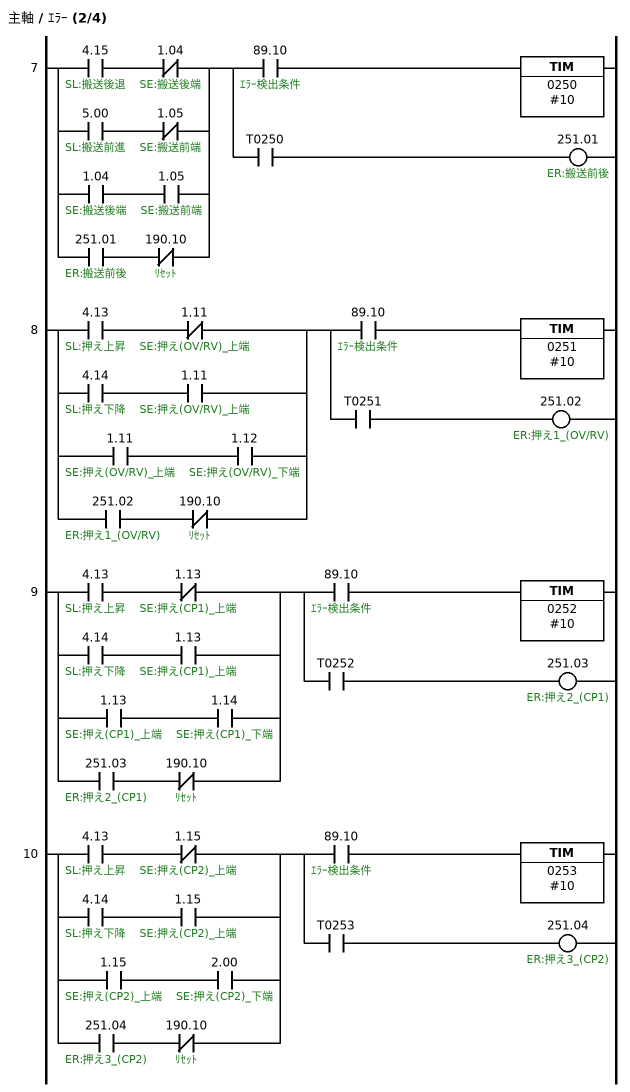
; rung 7
LD 4.15  ; SL:搬送後退
ANDNOT 1.04  ; SE:搬送後端
LD 5.00  ; SL:搬送前進
ANDNOT 1.05  ; SE:搬送前端
ORLD
LD 1.04  ; SE:搬送後端
AND 1.05  ; SE:搬送前端
ORLD
LD 251.01  ; ER:搬送前後
ANDNOT 190.10  ; ﾘｾｯﾄ
ORLD
OUT TR0
AND 89.10  ; ｴﾗｰ検出条件
TIM 0250 #10
LD TR0
AND T0250
OUT 251.01  ; ER:搬送前後
; rung 8
LD 4.13  ; SL:押え上昇
ANDNOT 1.11  ; SE:押え(OV/RV)_上端
LD 4.14  ; SL:押え下降
AND 1.11  ; SE:押え(OV/RV)_上端
ORLD
LD 1.11  ; SE:押え(OV/RV)_上端
AND 1.12  ; SE:押え(OV/RV)_下端
ORLD
LD 251.02  ; ER:押え1_(OV/RV)
ANDNOT 190.10  ; ﾘｾｯﾄ
ORLD
OUT TR0
AND 89.10  ; ｴﾗｰ検出条件
TIM 0251 #10
LD TR0
AND T0251
OUT 251.02  ; ER:押え1_(OV/RV)
; rung 9
LD 4.13  ; SL:押え上昇
ANDNOT 1.13  ; SE:押え(CP1)_上端
LD 4.14  ; SL:押え下降
AND 1.13  ; SE:押え(CP1)_上端
ORLD
LD 1.13  ; SE:押え(CP1)_上端
AND 1.14  ; SE:押え(CP1)_下端
ORLD
LD 251.03  ; ER:押え2_(CP1)
ANDNOT 190.10  ; ﾘｾｯﾄ
ORLD
OUT TR0
AND 89.10  ; ｴﾗｰ検出条件
TIM 0252 #10
LD TR0
AND T0252
OUT 251.03  ; ER:押え2_(CP1)
; rung 10
LD 4.13  ; SL:押え上昇
ANDNOT 1.15  ; SE:押え(CP2)_上端
LD 4.14  ; SL:押え下降
AND 1.15  ; SE:押え(CP2)_上端
ORLD
LD 1.15  ; SE:押え(CP2)_上端
AND 2.00  ; SE:押え(CP2)_下端
ORLD
LD 251.04  ; ER:押え3_(CP2)
ANDNOT 190.10  ; ﾘｾｯﾄ
ORLD
OUT TR0
AND 89.10  ; ｴﾗｰ検出条件
TIM 0253 #10
LD TR0
AND T0253
OUT 251.04  ; ER:押え3_(CP2)

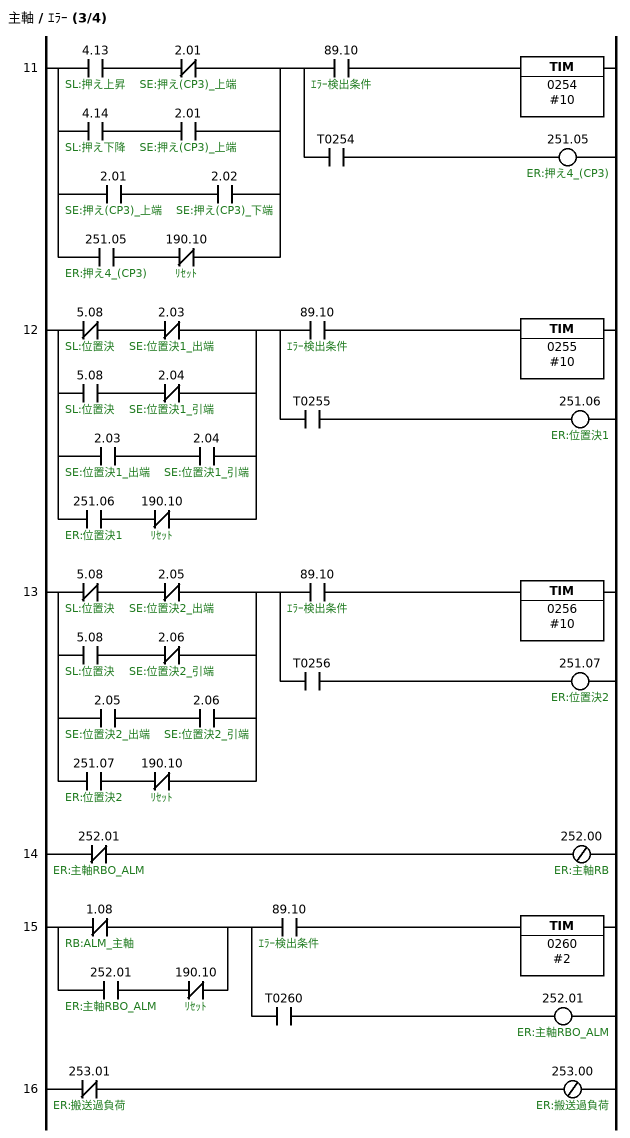
; rung 11
LD 4.13  ; SL:押え上昇
ANDNOT 2.01  ; SE:押え(CP3)_上端
LD 4.14  ; SL:押え下降
AND 2.01  ; SE:押え(CP3)_上端
ORLD
LD 2.01  ; SE:押え(CP3)_上端
AND 2.02  ; SE:押え(CP3)_下端
ORLD
LD 251.05  ; ER:押え4_(CP3)
ANDNOT 190.10  ; ﾘｾｯﾄ
ORLD
OUT TR0
AND 89.10  ; ｴﾗｰ検出条件
TIM 0254 #10
LD TR0
AND T0254
OUT 251.05  ; ER:押え4_(CP3)
; rung 12
LDNOT 5.08  ; SL:位置決
ANDNOT 2.03  ; SE:位置決1_出端
LD 5.08  ; SL:位置決
ANDNOT 2.04  ; SE:位置決1_引端
ORLD
LD 2.03  ; SE:位置決1_出端
AND 2.04  ; SE:位置決1_引端
ORLD
LD 251.06  ; ER:位置決1
ANDNOT 190.10  ; ﾘｾｯﾄ
ORLD
OUT TR0
AND 89.10  ; ｴﾗｰ検出条件
TIM 0255 #10
LD TR0
AND T0255
OUT 251.06  ; ER:位置決1
; rung 13
LDNOT 5.08  ; SL:位置決
ANDNOT 2.05  ; SE:位置決2_出端
LD 5.08  ; SL:位置決
ANDNOT 2.06  ; SE:位置決2_引端
ORLD
LD 2.05  ; SE:位置決2_出端
AND 2.06  ; SE:位置決2_引端
ORLD
LD 251.07  ; ER:位置決2
ANDNOT 190.10  ; ﾘｾｯﾄ
ORLD
OUT TR0
AND 89.10  ; ｴﾗｰ検出条件
TIM 0256 #10
LD TR0
AND T0256
OUT 251.07  ; ER:位置決2
; rung 14
LDNOT 252.01  ; ER:主軸RBO_ALM
OUTNOT 252.00  ; ER:主軸RB
; rung 15
LDNOT 1.08  ; RB:ALM_主軸
LD 252.01  ; ER:主軸RBO_ALM
ANDNOT 190.10  ; ﾘｾｯﾄ
ORLD
OUT TR0
AND 89.10  ; ｴﾗｰ検出条件
TIM 0260 #2
LD TR0
AND T0260
OUT 252.01  ; ER:主軸RBO_ALM
; rung 16
LDNOT 253.01  ; ER:搬送過負荷
OUTNOT 253.00  ; ER:搬送過負荷

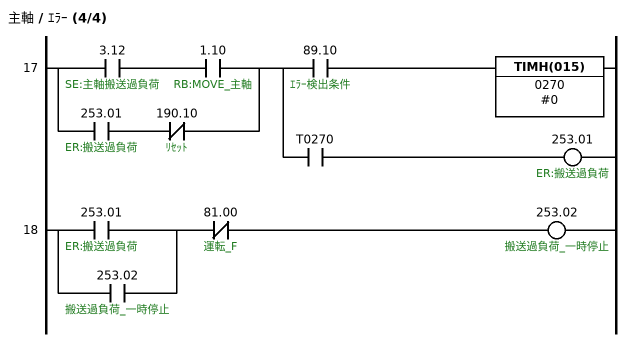
; rung 17
LD 3.12  ; SE:主軸搬送過負荷
AND 1.10  ; RB:MOVE_主軸
LD 253.01  ; ER:搬送過負荷
ANDNOT 190.10  ; ﾘｾｯﾄ
ORLD
OUT TR0
AND 89.10  ; ｴﾗｰ検出条件
TIMH(015) 0270 #0
LD TR0
AND T0270
OUT 253.01  ; ER:搬送過負荷
; rung 18
LD 253.01  ; ER:搬送過負荷
OR 253.02  ; 搬送過負荷_一時停止
ANDNOT 81.00  ; 運転_F
OUT 253.02  ; 搬送過負荷_一時停止

### Section END
; rung 0
END(001)

## Program 供給 (cyclic task 3)

### Section 制御

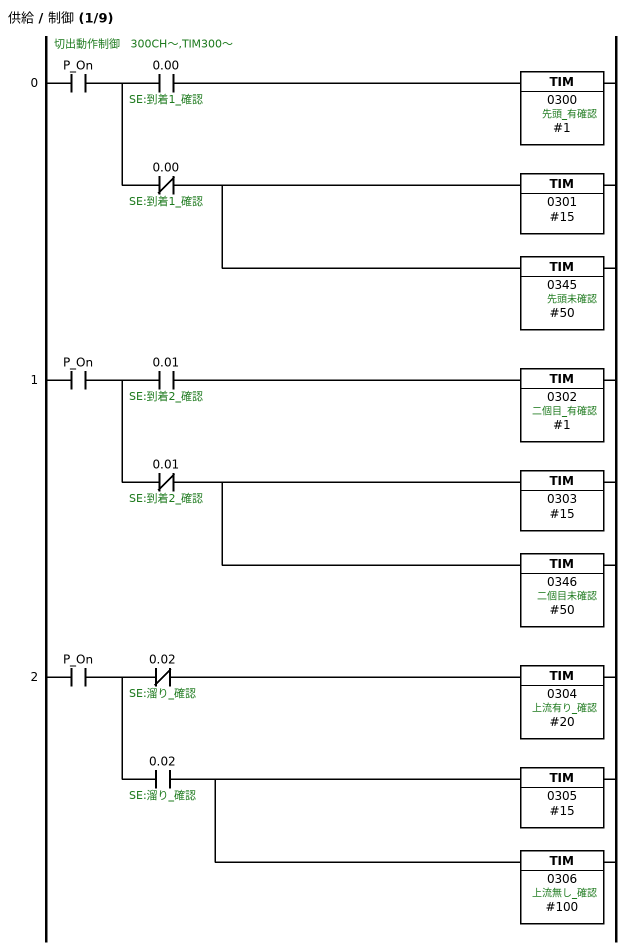
; rung 0: 切出動作制御   300CH～,TIM300～
LD P_On
OUT TR0
AND 0.00  ; SE:到着1_確認
TIM 0300 #1  ; 先頭_有確認
LD TR0
ANDNOT 0.00  ; SE:到着1_確認
TIM 0301 #15
TIM 0345 #50  ; 先頭未確認
; rung 1
LD P_On
OUT TR0
AND 0.01  ; SE:到着2_確認
TIM 0302 #1  ; 二個目_有確認
LD TR0
ANDNOT 0.01  ; SE:到着2_確認
TIM 0303 #15
TIM 0346 #50  ; 二個目未確認
; rung 2
LD P_On
OUT TR0
ANDNOT 0.02  ; SE:溜り_確認
TIM 0304 #20  ; 上流有り_確認
LD TR0
AND 0.02  ; SE:溜り_確認
TIM 0305 #15
TIM 0306 #100  ; 上流無し_確認

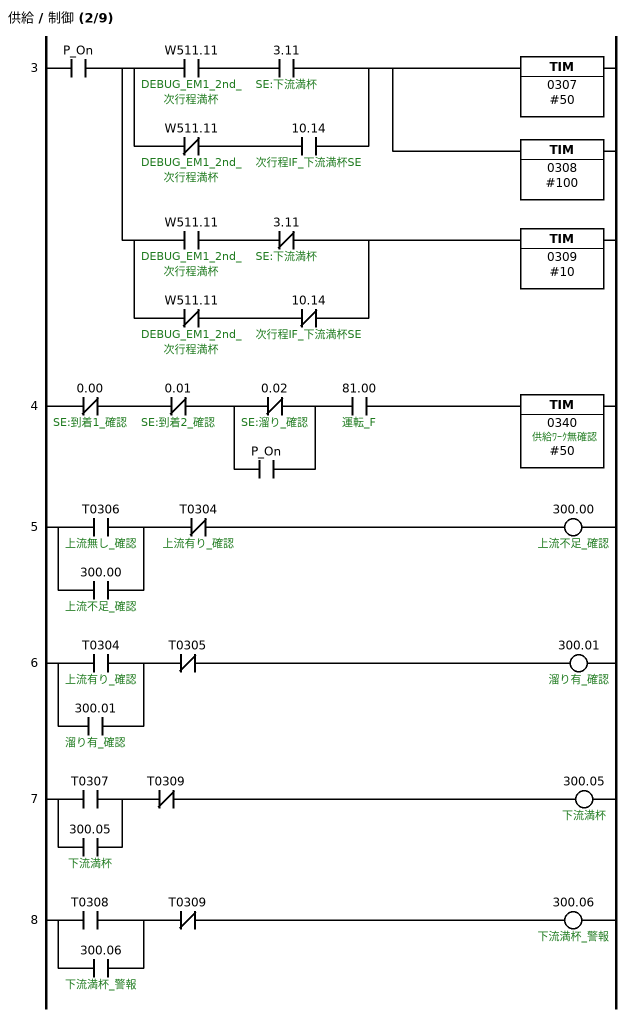
; rung 3
LD P_On
OUT TR0
LD W511.11  ; DEBUG_EM1_2nd_次行程満杯
AND 3.11  ; SE:下流満杯
LDNOT W511.11  ; DEBUG_EM1_2nd_次行程満杯
AND 10.14  ; 次行程IF_下流満杯SE
ORLD
ANDLD
TIM 0307 #50
TIM 0308 #100
LD TR0
LD W511.11  ; DEBUG_EM1_2nd_次行程満杯
ANDNOT 3.11  ; SE:下流満杯
LDNOT W511.11  ; DEBUG_EM1_2nd_次行程満杯
ANDNOT 10.14  ; 次行程IF_下流満杯SE
ORLD
ANDLD
TIM 0309 #10
; rung 4
LDNOT 0.00  ; SE:到着1_確認
ANDNOT 0.01  ; SE:到着2_確認
LDNOT 0.02  ; SE:溜り_確認
OR P_On
ANDLD
AND 81.00  ; 運転_F
TIM 0340 #50  ; 供給ﾜｰｸ無確認
; rung 5
LD T0306  ; 上流無し_確認
OR 300.00  ; 上流不足_確認
ANDNOT T0304  ; 上流有り_確認
OUT 300.00  ; 上流不足_確認
; rung 6
LD T0304  ; 上流有り_確認
OR 300.01  ; 溜り有_確認
ANDNOT T0305
OUT 300.01  ; 溜り有_確認
; rung 7
LD T0307
OR 300.05  ; 下流満杯
ANDNOT T0309
OUT 300.05  ; 下流満杯
; rung 8
LD T0308
OR 300.06  ; 下流満杯_警報
ANDNOT T0309
OUT 300.06  ; 下流満杯_警報

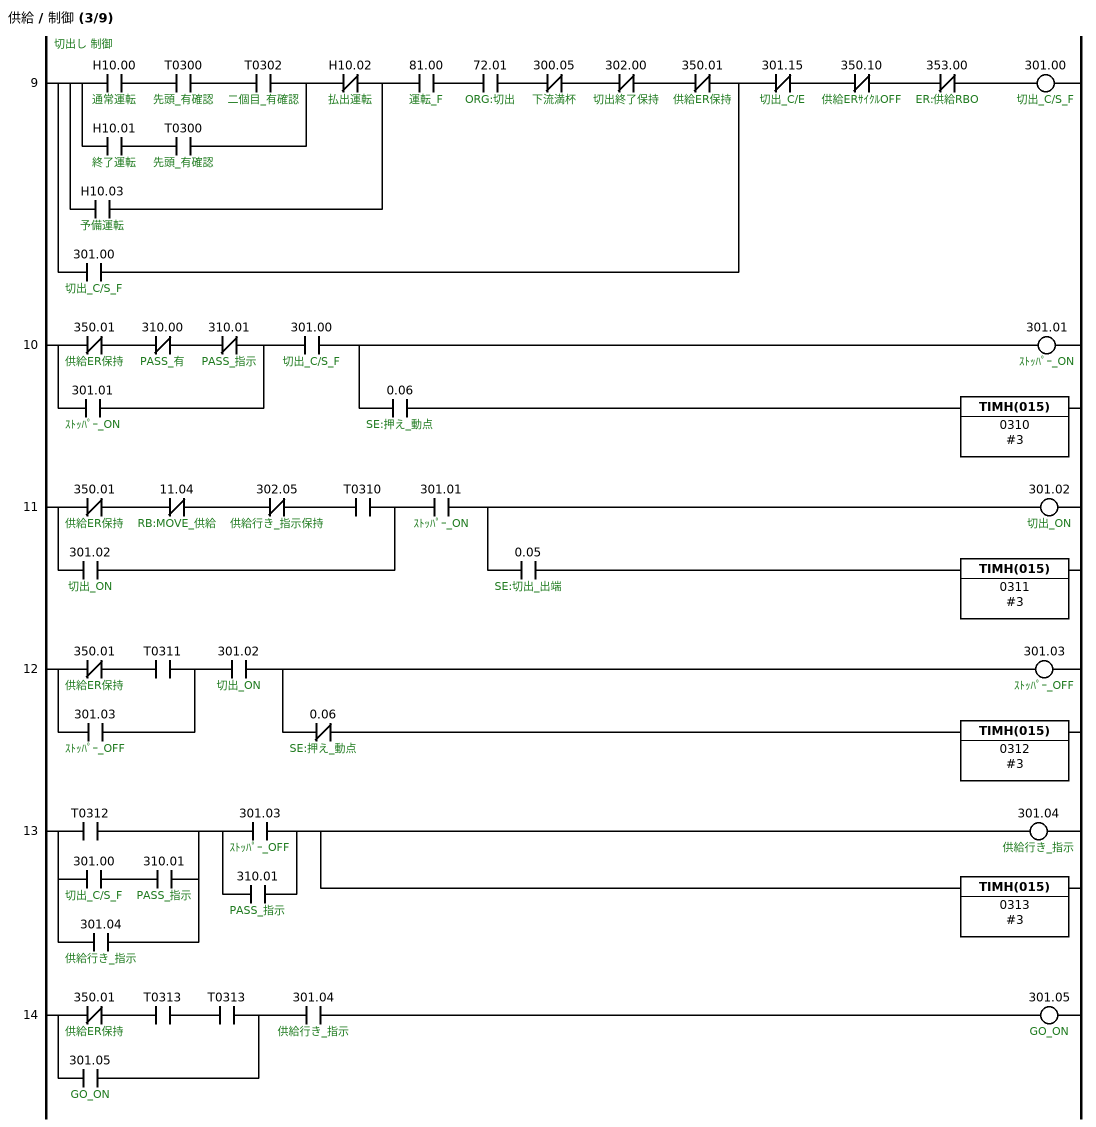
; rung 9: 切出し 制御
LD H10.00  ; 通常運転
AND T0300  ; 先頭_有確認
AND T0302  ; 二個目_有確認
LD H10.01  ; 終了運転
AND T0300  ; 先頭_有確認
ORLD
ANDNOT H10.02  ; 払出運転
OR H10.03  ; 予備運転
AND 81.00  ; 運転_F
AND 72.01  ; ORG:切出
ANDNOT 300.05  ; 下流満杯
ANDNOT 302.00  ; 切出終了保持
ANDNOT 350.01  ; 供給ER保持
OR 301.00  ; 切出_C/S_F
ANDNOT 301.15  ; 切出_C/E
ANDNOT 350.10  ; 供給ERｻｲｸﾙOFF
ANDNOT 353.00  ; ER:供給RBO
OUT 301.00  ; 切出_C/S_F
; rung 10
LDNOT 350.01  ; 供給ER保持
ANDNOT 310.00  ; PASS_有
ANDNOT 310.01  ; PASS_指示
OR 301.01  ; ｽﾄｯﾊﾟｰ_ON
AND 301.00  ; 切出_C/S_F
OUT 301.01  ; ｽﾄｯﾊﾟｰ_ON
AND 0.06  ; SE:押え_動点
TIMH(015) 0310 #3
; rung 11
LDNOT 350.01  ; 供給ER保持
ANDNOT 11.04  ; RB:MOVE_供給
ANDNOT 302.05  ; 供給行き_指示保持
AND T0310
OR 301.02  ; 切出_ON
AND 301.01  ; ｽﾄｯﾊﾟｰ_ON
OUT 301.02  ; 切出_ON
AND 0.05  ; SE:切出_出端
TIMH(015) 0311 #3
; rung 12
LDNOT 350.01  ; 供給ER保持
AND T0311
OR 301.03  ; ｽﾄｯﾊﾟｰ_OFF
AND 301.02  ; 切出_ON
OUT 301.03  ; ｽﾄｯﾊﾟｰ_OFF
ANDNOT 0.06  ; SE:押え_動点
TIMH(015) 0312 #3
; rung 13
LD T0312
LD 301.00  ; 切出_C/S_F
AND 310.01  ; PASS_指示
ORLD
OR 301.04  ; 供給行き_指示
LD 301.03  ; ｽﾄｯﾊﾟｰ_OFF
OR 310.01  ; PASS_指示
ANDLD
OUT 301.04  ; 供給行き_指示
TIMH(015) 0313 #3
; rung 14
LDNOT 350.01  ; 供給ER保持
AND T0313
AND T0313
OR 301.05  ; GO_ON
AND 301.04  ; 供給行き_指示
OUT 301.05  ; GO_ON

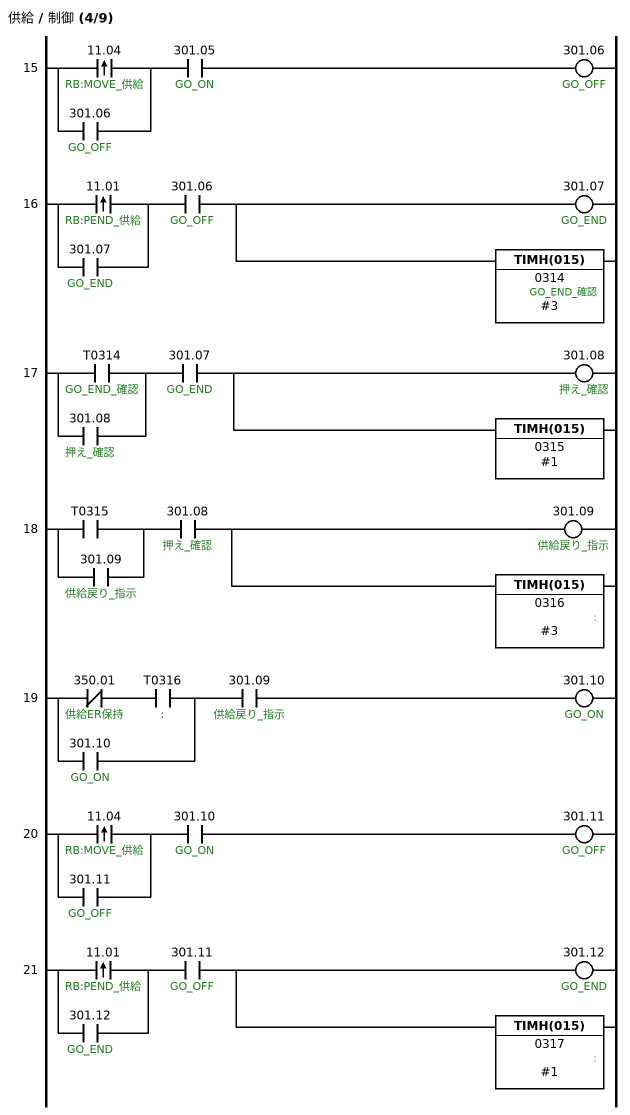
; rung 15
@LD 11.04  ; RB:MOVE_供給
OR 301.06  ; GO_OFF
AND 301.05  ; GO_ON
OUT 301.06  ; GO_OFF
; rung 16
@LD 11.01  ; RB:PEND_供給
OR 301.07  ; GO_END
AND 301.06  ; GO_OFF
OUT 301.07  ; GO_END
TIMH(015) 0314 #3  ; GO_END_確認
; rung 17
LD T0314  ; GO_END_確認
OR 301.08  ; 押え_確認
AND 301.07  ; GO_END
OUT 301.08  ; 押え_確認
TIMH(015) 0315 #1
; rung 18
LD T0315
OR 301.09  ; 供給戻り_指示
AND 301.08  ; 押え_確認
OUT 301.09  ; 供給戻り_指示
TIMH(015) 0316 #3  ; :
; rung 19
LDNOT 350.01  ; 供給ER保持
AND T0316  ; :
OR 301.10  ; GO_ON
AND 301.09  ; 供給戻り_指示
OUT 301.10  ; GO_ON
; rung 20
@LD 11.04  ; RB:MOVE_供給
OR 301.11  ; GO_OFF
AND 301.10  ; GO_ON
OUT 301.11  ; GO_OFF
; rung 21
@LD 11.01  ; RB:PEND_供給
OR 301.12  ; GO_END
AND 301.11  ; GO_OFF
OUT 301.12  ; GO_END
TIMH(015) 0317 #1  ; :

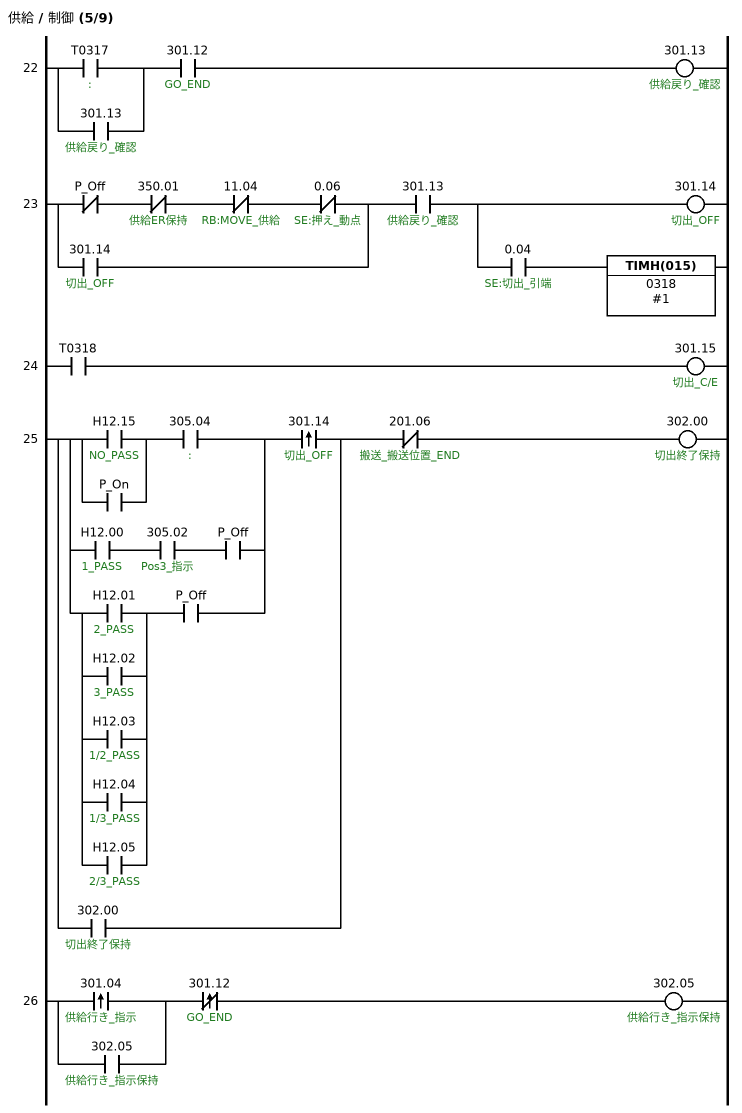
; rung 22
LD T0317  ; :
OR 301.13  ; 供給戻り_確認
AND 301.12  ; GO_END
OUT 301.13  ; 供給戻り_確認
; rung 23
LDNOT P_Off
ANDNOT 350.01  ; 供給ER保持
ANDNOT 11.04  ; RB:MOVE_供給
ANDNOT 0.06  ; SE:押え_動点
OR 301.14  ; 切出_OFF
AND 301.13  ; 供給戻り_確認
OUT 301.14  ; 切出_OFF
AND 0.04  ; SE:切出_引端
TIMH(015) 0318 #1
; rung 24
LD T0318
OUT 301.15  ; 切出_C/E
; rung 25
LD H12.15  ; NO_PASS
OR P_On
AND 305.04  ; :
LD H12.00  ; 1_PASS
AND 305.02  ; Pos3_指示
AND P_Off
ORLD
LD H12.01  ; 2_PASS
OR H12.02  ; 3_PASS
OR H12.03  ; 1/2_PASS
OR H12.04  ; 1/3_PASS
OR H12.05  ; 2/3_PASS
AND P_Off
ORLD
@AND 301.14  ; 切出_OFF
OR 302.00  ; 切出終了保持
ANDNOT 201.06  ; 搬送_搬送位置_END
OUT 302.00  ; 切出終了保持
; rung 26
@LD 301.04  ; 供給行き_指示
OR 302.05  ; 供給行き_指示保持
@ANDNOT 301.12  ; GO_END
OUT 302.05  ; 供給行き_指示保持

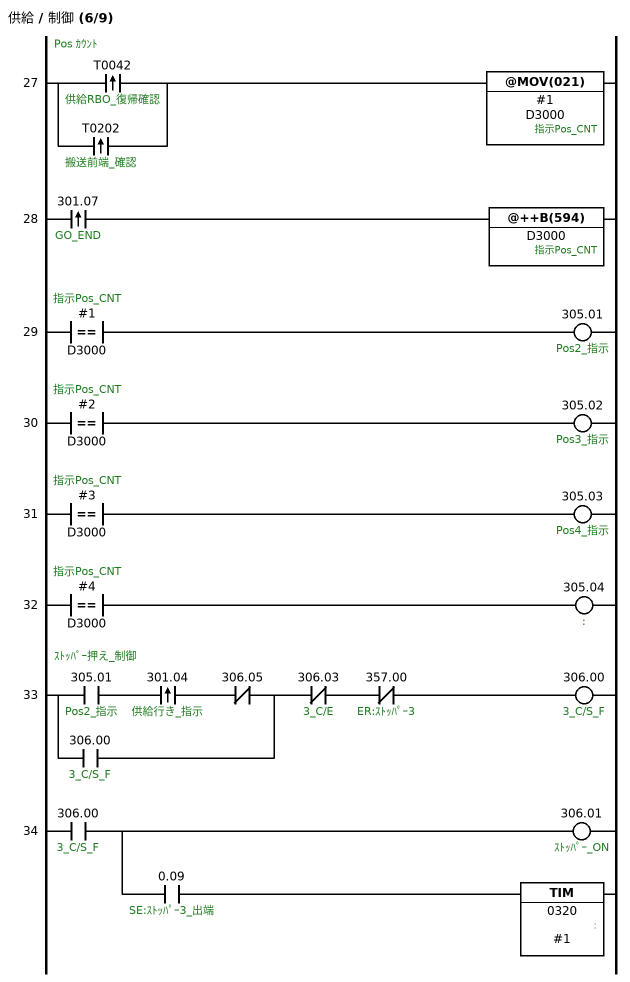
; rung 27: Pos ｶｳﾝﾄ
@LD T0042  ; 供給RBO_復帰確認
@OR T0202  ; 搬送前端_確認
@MOV(021) #1 D3000  ; 指示Pos_CNT
; rung 28
@LD 301.07  ; GO_END
@++B(594) D3000  ; 指示Pos_CNT
; rung 29
LD=(300) #1 D3000  ; 指示Pos_CNT
OUT 305.01  ; Pos2_指示
; rung 30
LD=(300) #2 D3000  ; 指示Pos_CNT
OUT 305.02  ; Pos3_指示
; rung 31
LD=(300) #3 D3000  ; 指示Pos_CNT
OUT 305.03  ; Pos4_指示
; rung 32
LD=(300) #4 D3000  ; 指示Pos_CNT
OUT 305.04  ; :
; rung 33: ｽﾄｯﾊﾟｰ押え_制御
LD 305.01  ; Pos2_指示
@AND 301.04  ; 供給行き_指示
ANDNOT 306.05
OR 306.00  ; 3_C/S_F
ANDNOT 306.03  ; 3_C/E
ANDNOT 357.00  ; ER:ｽﾄｯﾊﾟｰ3
OUT 306.00  ; 3_C/S_F
; rung 34
LD 306.00  ; 3_C/S_F
OUT 306.01  ; ｽﾄｯﾊﾟｰ_ON
AND 0.09  ; SE:ｽﾄｯﾊﾟｰ3_出端
TIM 0320 #1  ; :

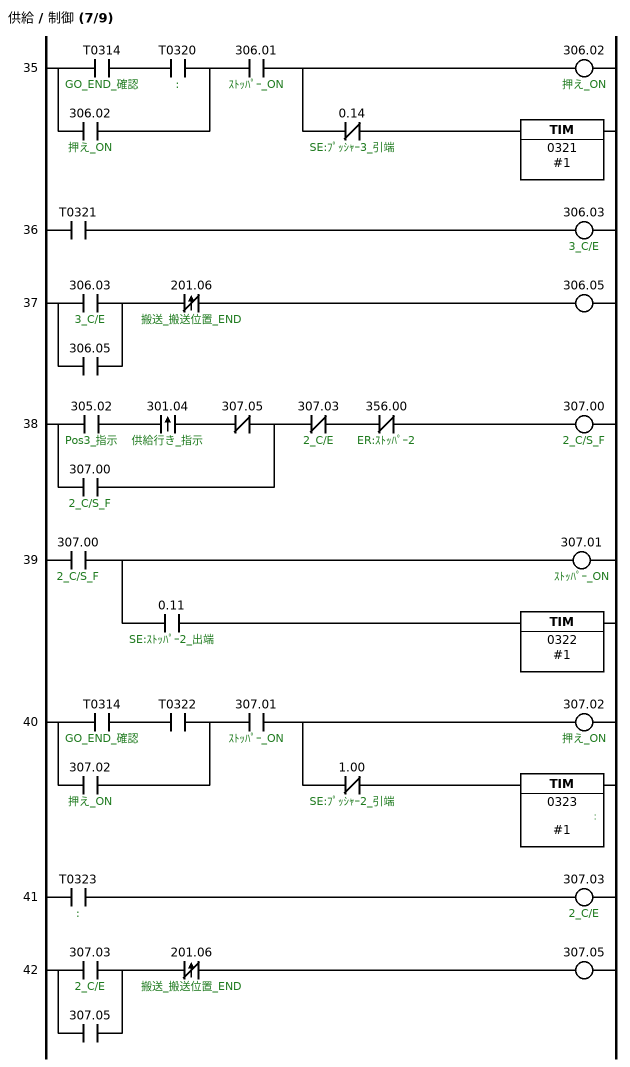
; rung 35
LD T0314  ; GO_END_確認
AND T0320  ; :
OR 306.02  ; 押え_ON
AND 306.01  ; ｽﾄｯﾊﾟｰ_ON
OUT 306.02  ; 押え_ON
ANDNOT 0.14  ; SE:ﾌﾟｯｼｬｰ3_引端
TIM 0321 #1
; rung 36
LD T0321
OUT 306.03  ; 3_C/E
; rung 37
LD 306.03  ; 3_C/E
OR 306.05
@ANDNOT 201.06  ; 搬送_搬送位置_END
OUT 306.05
; rung 38
LD 305.02  ; Pos3_指示
@AND 301.04  ; 供給行き_指示
ANDNOT 307.05
OR 307.00  ; 2_C/S_F
ANDNOT 307.03  ; 2_C/E
ANDNOT 356.00  ; ER:ｽﾄｯﾊﾟｰ2
OUT 307.00  ; 2_C/S_F
; rung 39
LD 307.00  ; 2_C/S_F
OUT 307.01  ; ｽﾄｯﾊﾟｰ_ON
AND 0.11  ; SE:ｽﾄｯﾊﾟｰ2_出端
TIM 0322 #1
; rung 40
LD T0314  ; GO_END_確認
AND T0322
OR 307.02  ; 押え_ON
AND 307.01  ; ｽﾄｯﾊﾟｰ_ON
OUT 307.02  ; 押え_ON
ANDNOT 1.00  ; SE:ﾌﾟｯｼｬｰ2_引端
TIM 0323 #1  ; :
; rung 41
LD T0323  ; :
OUT 307.03  ; 2_C/E
; rung 42
LD 307.03  ; 2_C/E
OR 307.05
@ANDNOT 201.06  ; 搬送_搬送位置_END
OUT 307.05

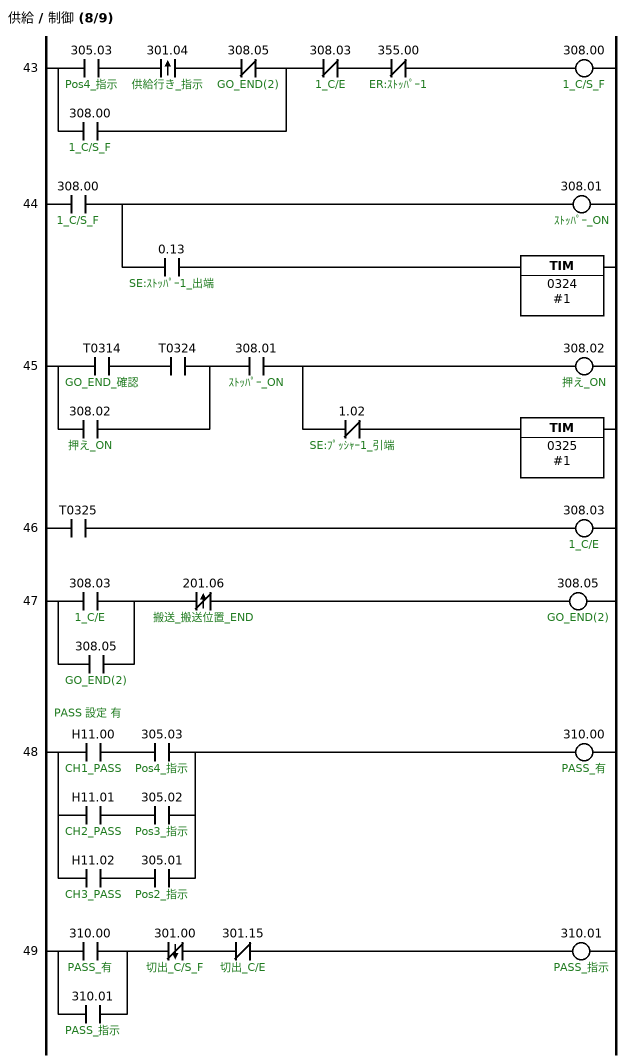
; rung 43
LD 305.03  ; Pos4_指示
@AND 301.04  ; 供給行き_指示
ANDNOT 308.05  ; GO_END(2)
OR 308.00  ; 1_C/S_F
ANDNOT 308.03  ; 1_C/E
ANDNOT 355.00  ; ER:ｽﾄｯﾊﾟｰ1
OUT 308.00  ; 1_C/S_F
; rung 44
LD 308.00  ; 1_C/S_F
OUT 308.01  ; ｽﾄｯﾊﾟｰ_ON
AND 0.13  ; SE:ｽﾄｯﾊﾟｰ1_出端
TIM 0324 #1
; rung 45
LD T0314  ; GO_END_確認
AND T0324
OR 308.02  ; 押え_ON
AND 308.01  ; ｽﾄｯﾊﾟｰ_ON
OUT 308.02  ; 押え_ON
ANDNOT 1.02  ; SE:ﾌﾟｯｼｬｰ1_引端
TIM 0325 #1
; rung 46
LD T0325
OUT 308.03  ; 1_C/E
; rung 47
LD 308.03  ; 1_C/E
OR 308.05  ; GO_END(2)
@ANDNOT 201.06  ; 搬送_搬送位置_END
OUT 308.05  ; GO_END(2)
; rung 48: PASS 設定 有
LD H11.00  ; CH1_PASS
AND 305.03  ; Pos4_指示
LD H11.01  ; CH2_PASS
AND 305.02  ; Pos3_指示
ORLD
LD H11.02  ; CH3_PASS
AND 305.01  ; Pos2_指示
ORLD
OUT 310.00  ; PASS_有
; rung 49
LD 310.00  ; PASS_有
OR 310.01  ; PASS_指示
%ANDNOT 301.00  ; 切出_C/S_F
ANDNOT 301.15  ; 切出_C/E
OUT 310.01  ; PASS_指示

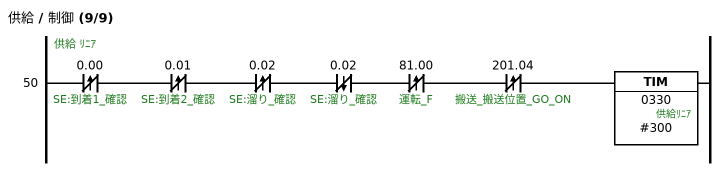
; rung 50: 供給 ﾘﾆｱ
@LDNOT 0.00  ; SE:到着1_確認
@ANDNOT 0.01  ; SE:到着2_確認
@ANDNOT 0.02  ; SE:溜り_確認
%ANDNOT 0.02  ; SE:溜り_確認
@ANDNOT 81.00  ; 運転_F
@ANDNOT 201.04  ; 搬送_搬送位置_GO_ON
TIM 0330 #300  ; 供給ﾘﾆｱ

### Section 出力

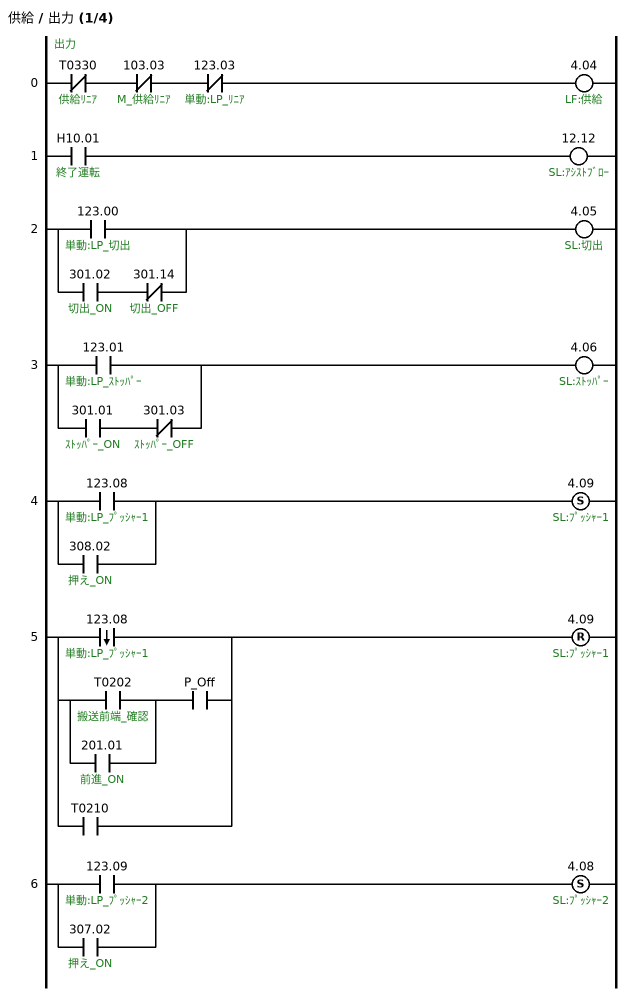
; rung 0: 出力
LDNOT T0330  ; 供給ﾘﾆｱ
ANDNOT 103.03  ; M_供給ﾘﾆｱ
ANDNOT 123.03  ; 単動:LP_ﾘﾆｱ
OUT 4.04  ; LF:供給
; rung 1
LD H10.01  ; 終了運転
OUT 12.12  ; SL:ｱｼｽﾄﾌﾞﾛｰ
; rung 2
LD 123.00  ; 単動:LP_切出
LD 301.02  ; 切出_ON
ANDNOT 301.14  ; 切出_OFF
ORLD
OUT 4.05  ; SL:切出
; rung 3
LD 123.01  ; 単動:LP_ｽﾄｯﾊﾟｰ
LD 301.01  ; ｽﾄｯﾊﾟｰ_ON
ANDNOT 301.03  ; ｽﾄｯﾊﾟｰ_OFF
ORLD
OUT 4.06  ; SL:ｽﾄｯﾊﾟｰ
; rung 4
LD 123.08  ; 単動:LP_ﾌﾟｯｼｬｰ1
OR 308.02  ; 押え_ON
SET 4.09  ; SL:ﾌﾟｯｼｬｰ1
; rung 5
%LD 123.08  ; 単動:LP_ﾌﾟｯｼｬｰ1
LD T0202  ; 搬送前端_確認
OR 201.01  ; 前進_ON
AND P_Off
ORLD
OR T0210
RSET 4.09  ; SL:ﾌﾟｯｼｬｰ1
; rung 6
LD 123.09  ; 単動:LP_ﾌﾟｯｼｬｰ2
OR 307.02  ; 押え_ON
SET 4.08  ; SL:ﾌﾟｯｼｬｰ2

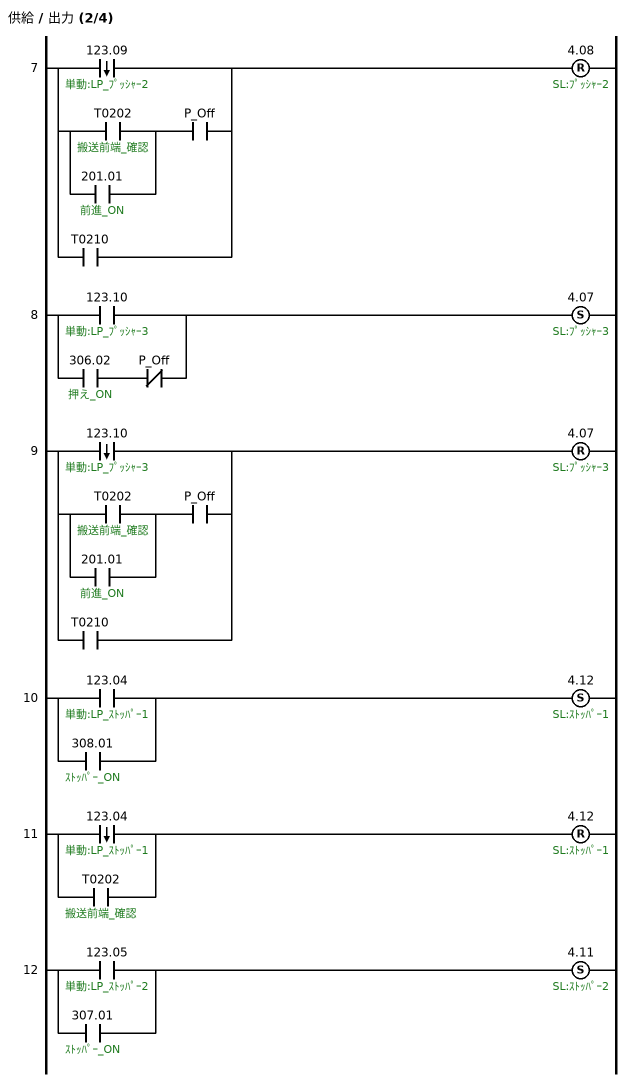
; rung 7
%LD 123.09  ; 単動:LP_ﾌﾟｯｼｬｰ2
LD T0202  ; 搬送前端_確認
OR 201.01  ; 前進_ON
AND P_Off
ORLD
OR T0210
RSET 4.08  ; SL:ﾌﾟｯｼｬｰ2
; rung 8
LD 123.10  ; 単動:LP_ﾌﾟｯｼｬｰ3
LD 306.02  ; 押え_ON
ANDNOT P_Off
ORLD
SET 4.07  ; SL:ﾌﾟｯｼｬｰ3
; rung 9
%LD 123.10  ; 単動:LP_ﾌﾟｯｼｬｰ3
LD T0202  ; 搬送前端_確認
OR 201.01  ; 前進_ON
AND P_Off
ORLD
OR T0210
RSET 4.07  ; SL:ﾌﾟｯｼｬｰ3
; rung 10
LD 123.04  ; 単動:LP_ｽﾄｯﾊﾟｰ1
OR 308.01  ; ｽﾄｯﾊﾟｰ_ON
SET 4.12  ; SL:ｽﾄｯﾊﾟｰ1
; rung 11
%LD 123.04  ; 単動:LP_ｽﾄｯﾊﾟｰ1
OR T0202  ; 搬送前端_確認
RSET 4.12  ; SL:ｽﾄｯﾊﾟｰ1
; rung 12
LD 123.05  ; 単動:LP_ｽﾄｯﾊﾟｰ2
OR 307.01  ; ｽﾄｯﾊﾟｰ_ON
SET 4.11  ; SL:ｽﾄｯﾊﾟｰ2

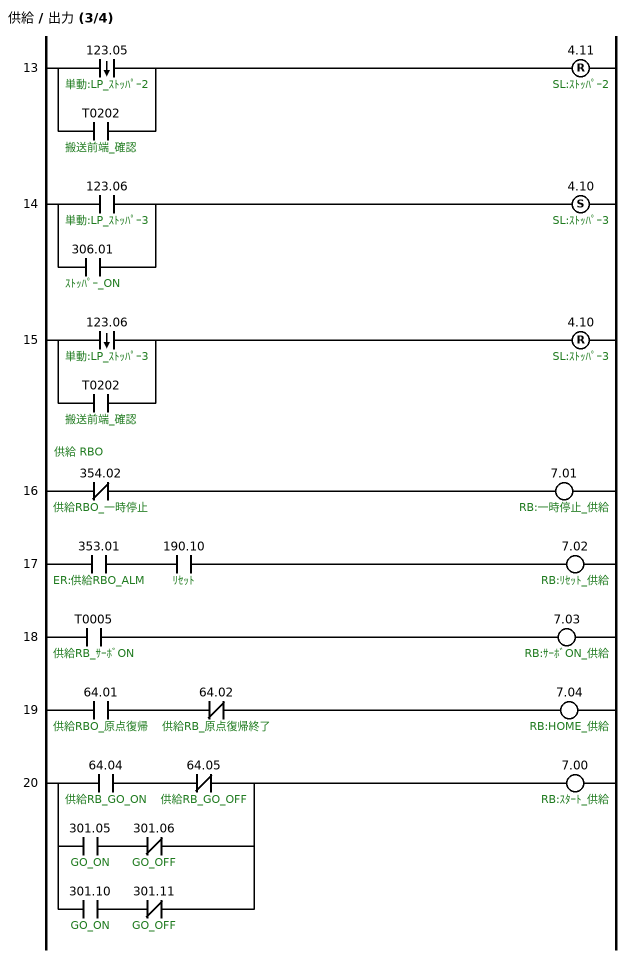
; rung 13
%LD 123.05  ; 単動:LP_ｽﾄｯﾊﾟｰ2
OR T0202  ; 搬送前端_確認
RSET 4.11  ; SL:ｽﾄｯﾊﾟｰ2
; rung 14
LD 123.06  ; 単動:LP_ｽﾄｯﾊﾟｰ3
OR 306.01  ; ｽﾄｯﾊﾟｰ_ON
SET 4.10  ; SL:ｽﾄｯﾊﾟｰ3
; rung 15
%LD 123.06  ; 単動:LP_ｽﾄｯﾊﾟｰ3
OR T0202  ; 搬送前端_確認
RSET 4.10  ; SL:ｽﾄｯﾊﾟｰ3
; rung 16: 供給 RBO
LDNOT 354.02  ; 供給RBO_一時停止
OUT 7.01  ; RB:一時停止_供給
; rung 17
LD 353.01  ; ER:供給RBO_ALM
AND 190.10  ; ﾘｾｯﾄ
OUT 7.02  ; RB:ﾘｾｯﾄ_供給
; rung 18
LD T0005  ; 供給RB_ｻｰﾎﾞON
OUT 7.03  ; RB:ｻｰﾎﾞON_供給
; rung 19
LD 64.01  ; 供給RBO_原点復帰
ANDNOT 64.02  ; 供給RB_原点復帰終了
OUT 7.04  ; RB:HOME_供給
; rung 20
LD 64.04  ; 供給RB_GO_ON
ANDNOT 64.05  ; 供給RB_GO_OFF
LD 301.05  ; GO_ON
ANDNOT 301.06  ; GO_OFF
ORLD
LD 301.10  ; GO_ON
ANDNOT 301.11  ; GO_OFF
ORLD
OUT 7.00  ; RB:ｽﾀｰﾄ_供給

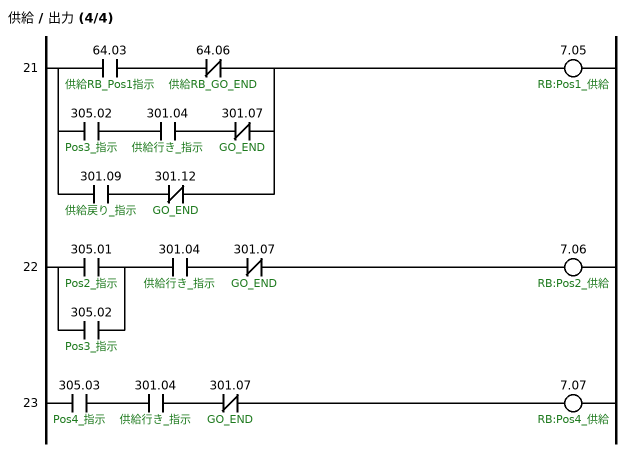
; rung 21
LD 64.03  ; 供給RB_Pos1指示
ANDNOT 64.06  ; 供給RB_GO_END
LD 305.02  ; Pos3_指示
AND 301.04  ; 供給行き_指示
ANDNOT 301.07  ; GO_END
ORLD
LD 301.09  ; 供給戻り_指示
ANDNOT 301.12  ; GO_END
ORLD
OUT 7.05  ; RB:Pos1_供給
; rung 22
LD 305.01  ; Pos2_指示
OR 305.02  ; Pos3_指示
AND 301.04  ; 供給行き_指示
ANDNOT 301.07  ; GO_END
OUT 7.06  ; RB:Pos2_供給
; rung 23
LD 305.03  ; Pos4_指示
AND 301.04  ; 供給行き_指示
ANDNOT 301.07  ; GO_END
OUT 7.07  ; RB:Pos4_供給

### Section ｴﾗｰ

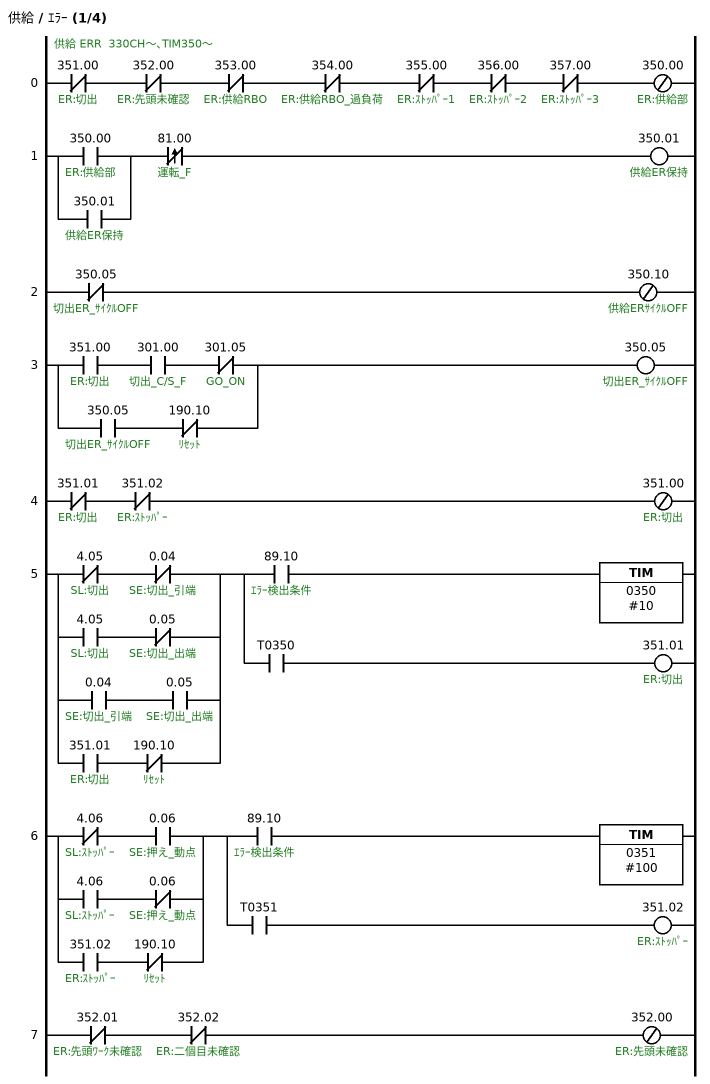
; rung 0: 供給 ERR  330CH～､TIM350～
LDNOT 351.00  ; ER:切出
ANDNOT 352.00  ; ER:先頭未確認
ANDNOT 353.00  ; ER:供給RBO
ANDNOT 354.00  ; ER:供給RBO_過負荷
ANDNOT 355.00  ; ER:ｽﾄｯﾊﾟｰ1
ANDNOT 356.00  ; ER:ｽﾄｯﾊﾟｰ2
ANDNOT 357.00  ; ER:ｽﾄｯﾊﾟｰ3
OUTNOT 350.00  ; ER:供給部
; rung 1
LD 350.00  ; ER:供給部
OR 350.01  ; 供給ER保持
@ANDNOT 81.00  ; 運転_F
OUT 350.01  ; 供給ER保持
; rung 2
LDNOT 350.05  ; 切出ER_ｻｲｸﾙOFF
OUTNOT 350.10  ; 供給ERｻｲｸﾙOFF
; rung 3
LD 351.00  ; ER:切出
AND 301.00  ; 切出_C/S_F
ANDNOT 301.05  ; GO_ON
LD 350.05  ; 切出ER_ｻｲｸﾙOFF
ANDNOT 190.10  ; ﾘｾｯﾄ
ORLD
OUT 350.05  ; 切出ER_ｻｲｸﾙOFF
; rung 4
LDNOT 351.01  ; ER:切出
ANDNOT 351.02  ; ER:ｽﾄｯﾊﾟｰ
OUTNOT 351.00  ; ER:切出
; rung 5
LDNOT 4.05  ; SL:切出
ANDNOT 0.04  ; SE:切出_引端
LD 4.05  ; SL:切出
ANDNOT 0.05  ; SE:切出_出端
ORLD
LD 0.04  ; SE:切出_引端
AND 0.05  ; SE:切出_出端
ORLD
LD 351.01  ; ER:切出
ANDNOT 190.10  ; ﾘｾｯﾄ
ORLD
OUT TR0
AND 89.10  ; ｴﾗｰ検出条件
TIM 0350 #10
LD TR0
AND T0350
OUT 351.01  ; ER:切出
; rung 6
LDNOT 4.06  ; SL:ｽﾄｯﾊﾟｰ
AND 0.06  ; SE:押え_動点
LD 4.06  ; SL:ｽﾄｯﾊﾟｰ
ANDNOT 0.06  ; SE:押え_動点
ORLD
LD 351.02  ; ER:ｽﾄｯﾊﾟｰ
ANDNOT 190.10  ; ﾘｾｯﾄ
ORLD
OUT TR0
AND 89.10  ; ｴﾗｰ検出条件
TIM 0351 #100
LD TR0
AND T0351
OUT 351.02  ; ER:ｽﾄｯﾊﾟｰ
; rung 7
LDNOT 352.01  ; ER:先頭ﾜｰｸ未確認
ANDNOT 352.02  ; ER:二個目未確認
OUTNOT 352.00  ; ER:先頭未確認

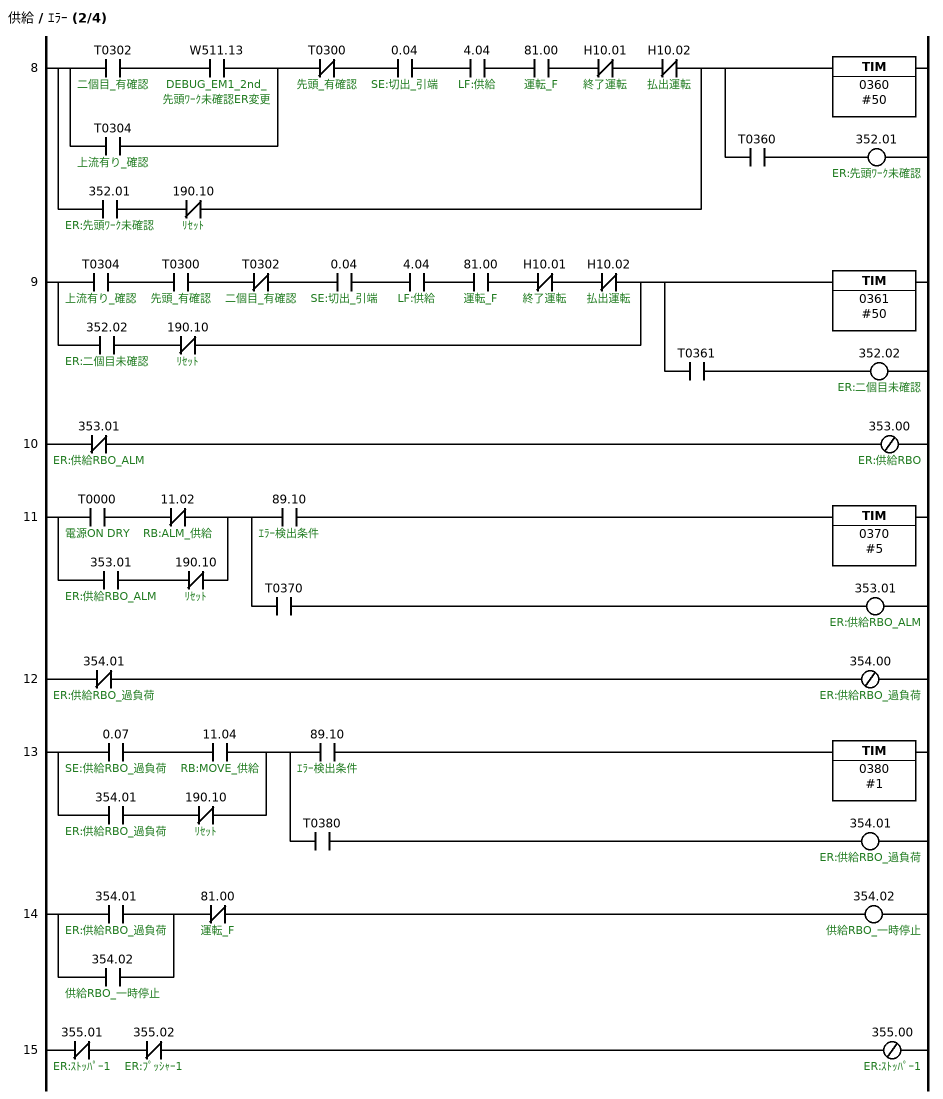
; rung 8
LD T0302  ; 二個目_有確認
AND W511.13  ; DEBUG_EM1_2nd_先頭ﾜｰｸ未確認ER変更
OR T0304  ; 上流有り_確認
ANDNOT T0300  ; 先頭_有確認
AND 0.04  ; SE:切出_引端
AND 4.04  ; LF:供給
AND 81.00  ; 運転_F
ANDNOT H10.01  ; 終了運転
ANDNOT H10.02  ; 払出運転
LD 352.01  ; ER:先頭ﾜｰｸ未確認
ANDNOT 190.10  ; ﾘｾｯﾄ
ORLD
TIM 0360 #50
AND T0360
OUT 352.01  ; ER:先頭ﾜｰｸ未確認
; rung 9
LD T0304  ; 上流有り_確認
AND T0300  ; 先頭_有確認
ANDNOT T0302  ; 二個目_有確認
AND 0.04  ; SE:切出_引端
AND 4.04  ; LF:供給
AND 81.00  ; 運転_F
ANDNOT H10.01  ; 終了運転
ANDNOT H10.02  ; 払出運転
LD 352.02  ; ER:二個目未確認
ANDNOT 190.10  ; ﾘｾｯﾄ
ORLD
TIM 0361 #50
AND T0361
OUT 352.02  ; ER:二個目未確認
; rung 10
LDNOT 353.01  ; ER:供給RBO_ALM
OUTNOT 353.00  ; ER:供給RBO
; rung 11
LD T0000  ; 電源ON DRY
ANDNOT 11.02  ; RB:ALM_供給
LD 353.01  ; ER:供給RBO_ALM
ANDNOT 190.10  ; ﾘｾｯﾄ
ORLD
OUT TR0
AND 89.10  ; ｴﾗｰ検出条件
TIM 0370 #5
LD TR0
AND T0370
OUT 353.01  ; ER:供給RBO_ALM
; rung 12
LDNOT 354.01  ; ER:供給RBO_過負荷
OUTNOT 354.00  ; ER:供給RBO_過負荷
; rung 13
LD 0.07  ; SE:供給RBO_過負荷
AND 11.04  ; RB:MOVE_供給
LD 354.01  ; ER:供給RBO_過負荷
ANDNOT 190.10  ; ﾘｾｯﾄ
ORLD
OUT TR0
AND 89.10  ; ｴﾗｰ検出条件
TIM 0380 #1
LD TR0
AND T0380
OUT 354.01  ; ER:供給RBO_過負荷
; rung 14
LD 354.01  ; ER:供給RBO_過負荷
OR 354.02  ; 供給RBO_一時停止
ANDNOT 81.00  ; 運転_F
OUT 354.02  ; 供給RBO_一時停止
; rung 15
LDNOT 355.01  ; ER:ｽﾄｯﾊﾟｰ1
ANDNOT 355.02  ; ER:ﾌﾟｯｼｬｰ1
OUTNOT 355.00  ; ER:ｽﾄｯﾊﾟｰ1

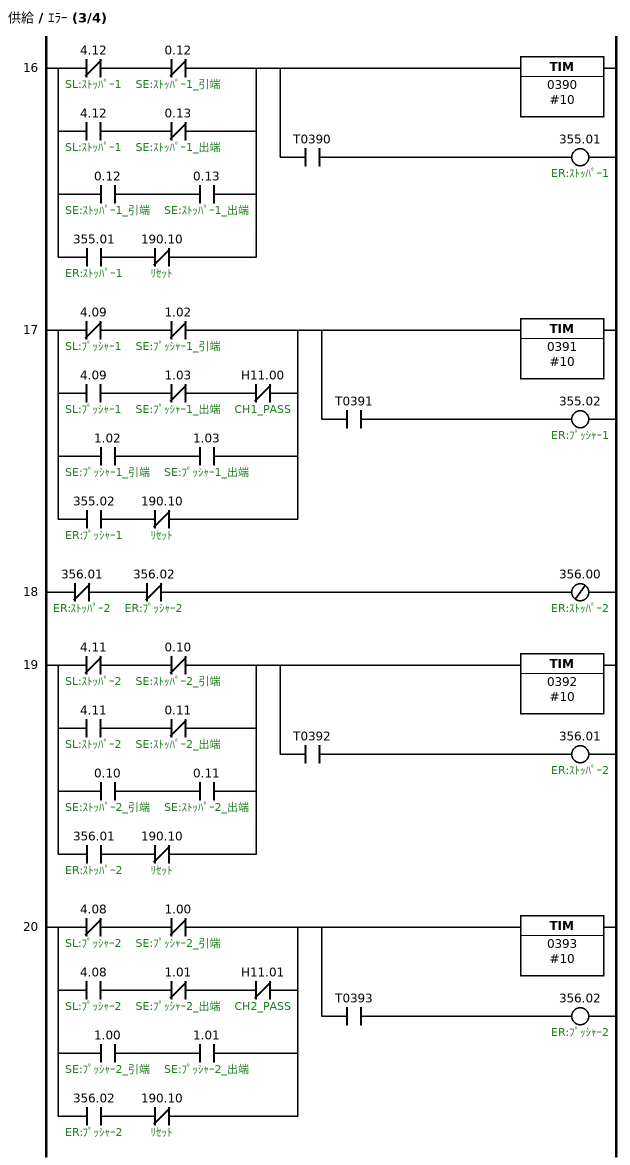
; rung 16
LDNOT 4.12  ; SL:ｽﾄｯﾊﾟｰ1
ANDNOT 0.12  ; SE:ｽﾄｯﾊﾟｰ1_引端
LD 4.12  ; SL:ｽﾄｯﾊﾟｰ1
ANDNOT 0.13  ; SE:ｽﾄｯﾊﾟｰ1_出端
ORLD
LD 0.12  ; SE:ｽﾄｯﾊﾟｰ1_引端
AND 0.13  ; SE:ｽﾄｯﾊﾟｰ1_出端
ORLD
LD 355.01  ; ER:ｽﾄｯﾊﾟｰ1
ANDNOT 190.10  ; ﾘｾｯﾄ
ORLD
TIM 0390 #10
AND T0390
OUT 355.01  ; ER:ｽﾄｯﾊﾟｰ1
; rung 17
LDNOT 4.09  ; SL:ﾌﾟｯｼｬｰ1
ANDNOT 1.02  ; SE:ﾌﾟｯｼｬｰ1_引端
LD 4.09  ; SL:ﾌﾟｯｼｬｰ1
ANDNOT 1.03  ; SE:ﾌﾟｯｼｬｰ1_出端
ANDNOT H11.00  ; CH1_PASS
ORLD
LD 1.02  ; SE:ﾌﾟｯｼｬｰ1_引端
AND 1.03  ; SE:ﾌﾟｯｼｬｰ1_出端
ORLD
LD 355.02  ; ER:ﾌﾟｯｼｬｰ1
ANDNOT 190.10  ; ﾘｾｯﾄ
ORLD
TIM 0391 #10
AND T0391
OUT 355.02  ; ER:ﾌﾟｯｼｬｰ1
; rung 18
LDNOT 356.01  ; ER:ｽﾄｯﾊﾟｰ2
ANDNOT 356.02  ; ER:ﾌﾟｯｼｬｰ2
OUTNOT 356.00  ; ER:ｽﾄｯﾊﾟｰ2
; rung 19
LDNOT 4.11  ; SL:ｽﾄｯﾊﾟｰ2
ANDNOT 0.10  ; SE:ｽﾄｯﾊﾟｰ2_引端
LD 4.11  ; SL:ｽﾄｯﾊﾟｰ2
ANDNOT 0.11  ; SE:ｽﾄｯﾊﾟｰ2_出端
ORLD
LD 0.10  ; SE:ｽﾄｯﾊﾟｰ2_引端
AND 0.11  ; SE:ｽﾄｯﾊﾟｰ2_出端
ORLD
LD 356.01  ; ER:ｽﾄｯﾊﾟｰ2
ANDNOT 190.10  ; ﾘｾｯﾄ
ORLD
TIM 0392 #10
AND T0392
OUT 356.01  ; ER:ｽﾄｯﾊﾟｰ2
; rung 20
LDNOT 4.08  ; SL:ﾌﾟｯｼｬｰ2
ANDNOT 1.00  ; SE:ﾌﾟｯｼｬｰ2_引端
LD 4.08  ; SL:ﾌﾟｯｼｬｰ2
ANDNOT 1.01  ; SE:ﾌﾟｯｼｬｰ2_出端
ANDNOT H11.01  ; CH2_PASS
ORLD
LD 1.00  ; SE:ﾌﾟｯｼｬｰ2_引端
AND 1.01  ; SE:ﾌﾟｯｼｬｰ2_出端
ORLD
LD 356.02  ; ER:ﾌﾟｯｼｬｰ2
ANDNOT 190.10  ; ﾘｾｯﾄ
ORLD
TIM 0393 #10
AND T0393
OUT 356.02  ; ER:ﾌﾟｯｼｬｰ2

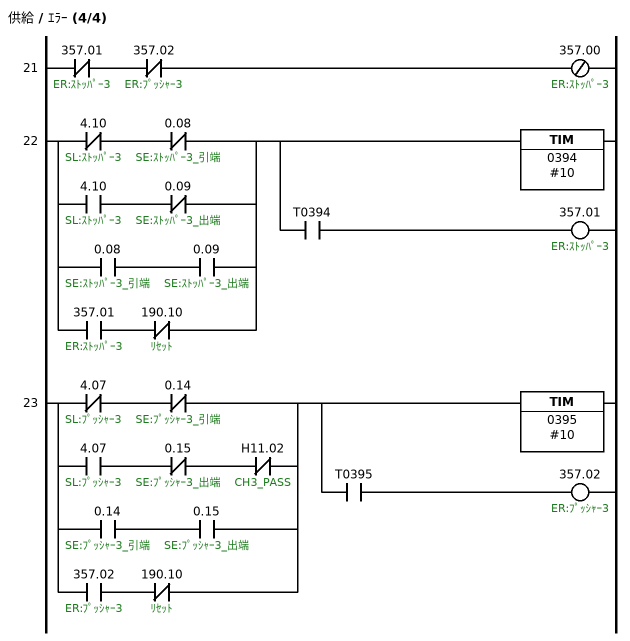
; rung 21
LDNOT 357.01  ; ER:ｽﾄｯﾊﾟｰ3
ANDNOT 357.02  ; ER:ﾌﾟｯｼｬｰ3
OUTNOT 357.00  ; ER:ｽﾄｯﾊﾟｰ3
; rung 22
LDNOT 4.10  ; SL:ｽﾄｯﾊﾟｰ3
ANDNOT 0.08  ; SE:ｽﾄｯﾊﾟｰ3_引端
LD 4.10  ; SL:ｽﾄｯﾊﾟｰ3
ANDNOT 0.09  ; SE:ｽﾄｯﾊﾟｰ3_出端
ORLD
LD 0.08  ; SE:ｽﾄｯﾊﾟｰ3_引端
AND 0.09  ; SE:ｽﾄｯﾊﾟｰ3_出端
ORLD
LD 357.01  ; ER:ｽﾄｯﾊﾟｰ3
ANDNOT 190.10  ; ﾘｾｯﾄ
ORLD
TIM 0394 #10
AND T0394
OUT 357.01  ; ER:ｽﾄｯﾊﾟｰ3
; rung 23
LDNOT 4.07  ; SL:ﾌﾟｯｼｬｰ3
ANDNOT 0.14  ; SE:ﾌﾟｯｼｬｰ3_引端
LD 4.07  ; SL:ﾌﾟｯｼｬｰ3
ANDNOT 0.15  ; SE:ﾌﾟｯｼｬｰ3_出端
ANDNOT H11.02  ; CH3_PASS
ORLD
LD 0.14  ; SE:ﾌﾟｯｼｬｰ3_引端
AND 0.15  ; SE:ﾌﾟｯｼｬｰ3_出端
ORLD
LD 357.02  ; ER:ﾌﾟｯｼｬｰ3
ANDNOT 190.10  ; ﾘｾｯﾄ
ORLD
TIM 0395 #10
AND T0395
OUT 357.02  ; ER:ﾌﾟｯｼｬｰ3

### Section END
; rung 0
END(001)

## Program 測定 (cyclic task 4)

### Section 制御

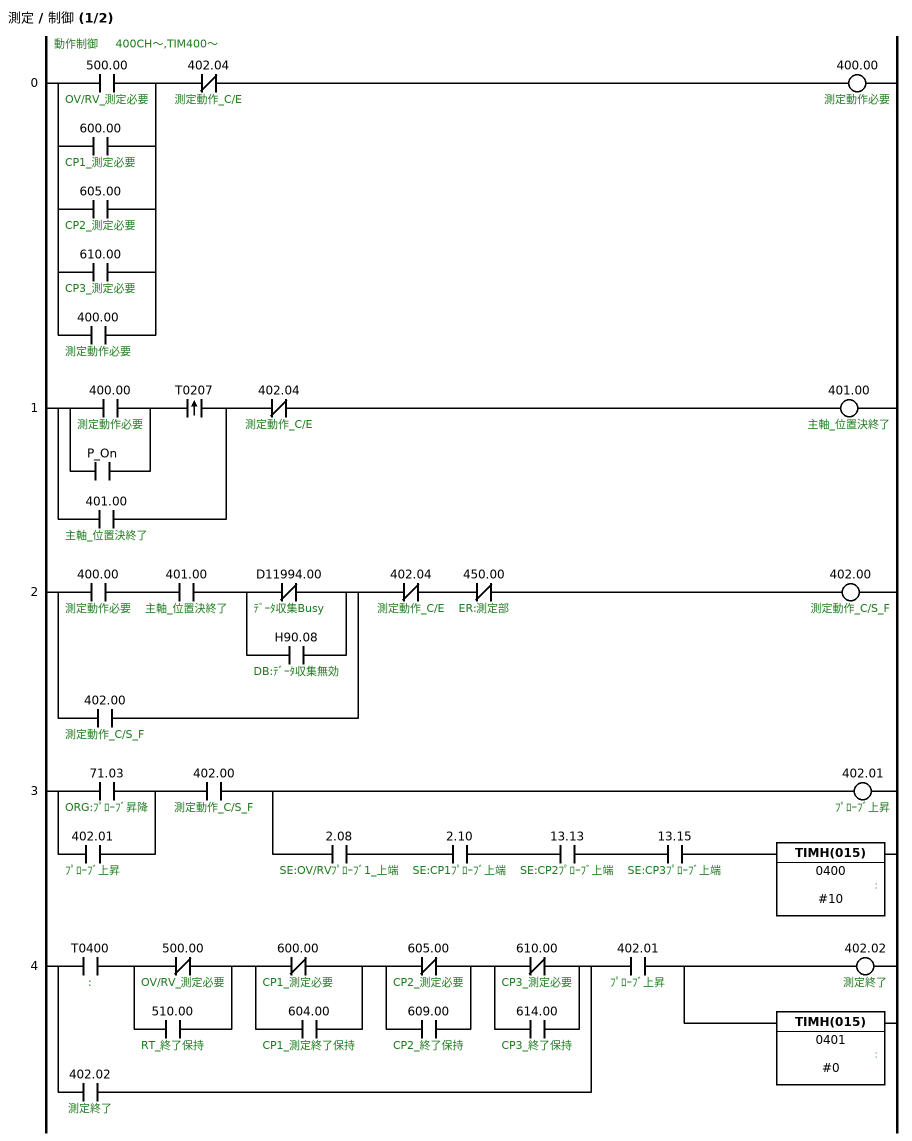
; rung 0: 動作制御     400CH～,TIM400～
LD 500.00  ; OV/RV_測定必要
OR 600.00  ; CP1_測定必要
OR 605.00  ; CP2_測定必要
OR 610.00  ; CP3_測定必要
OR 400.00  ; 測定動作必要
ANDNOT 402.04  ; 測定動作_C/E
OUT 400.00  ; 測定動作必要
; rung 1
LD 400.00  ; 測定動作必要
OR P_On
@AND T0207
OR 401.00  ; 主軸_位置決終了
ANDNOT 402.04  ; 測定動作_C/E
OUT 401.00  ; 主軸_位置決終了
; rung 2
LD 400.00  ; 測定動作必要
AND 401.00  ; 主軸_位置決終了
LDNOT D11994.00  ; ﾃﾞｰﾀ収集Busy
OR H90.08  ; DB:ﾃﾞｰﾀ収集無効
ANDLD
OR 402.00  ; 測定動作_C/S_F
ANDNOT 402.04  ; 測定動作_C/E
ANDNOT 450.00  ; ER:測定部
OUT 402.00  ; 測定動作_C/S_F
; rung 3
LD 71.03  ; ORG:ﾌﾟﾛｰﾌﾞ昇降
OR 402.01  ; ﾌﾟﾛｰﾌﾞ上昇
AND 402.00  ; 測定動作_C/S_F
OUT 402.01  ; ﾌﾟﾛｰﾌﾞ上昇
AND 2.08  ; SE:OV/RVﾌﾟﾛｰﾌﾞ1_上端
AND 2.10  ; SE:CP1ﾌﾟﾛｰﾌﾞ上端
AND 13.13  ; SE:CP2ﾌﾟﾛｰﾌﾞ上端
AND 13.15  ; SE:CP3ﾌﾟﾛｰﾌﾞ上端
TIMH(015) 0400 #10  ; :
; rung 4
LD T0400  ; :
LDNOT 500.00  ; OV/RV_測定必要
OR 510.00  ; RT_終了保持
ANDLD
LDNOT 600.00  ; CP1_測定必要
OR 604.00  ; CP1_測定終了保持
ANDLD
LDNOT 605.00  ; CP2_測定必要
OR 609.00  ; CP2_終了保持
ANDLD
LDNOT 610.00  ; CP3_測定必要
OR 614.00  ; CP3_終了保持
ANDLD
OR 402.02  ; 測定終了
AND 402.01  ; ﾌﾟﾛｰﾌﾞ上昇
OUT 402.02  ; 測定終了
TIMH(015) 0401 #0  ; :

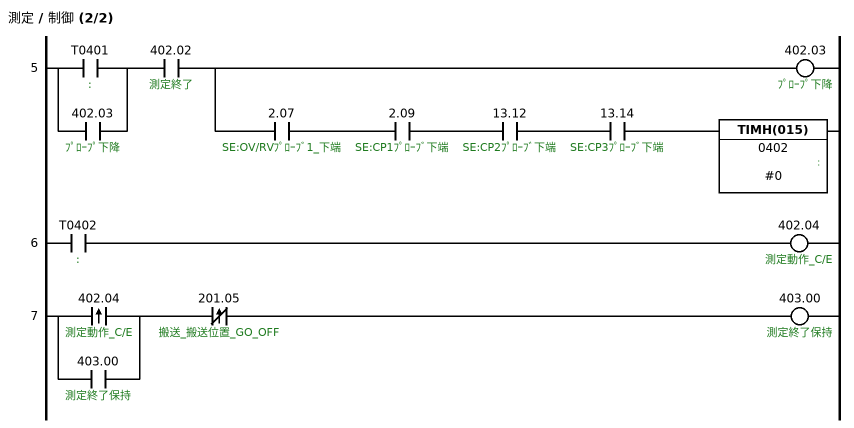
; rung 5
LD T0401  ; :
OR 402.03  ; ﾌﾟﾛｰﾌﾟ下降
AND 402.02  ; 測定終了
OUT 402.03  ; ﾌﾟﾛｰﾌﾟ下降
AND 2.07  ; SE:OV/RVﾌﾟﾛｰﾌﾞ1_下端
AND 2.09  ; SE:CP1ﾌﾟﾛｰﾌﾞ下端
AND 13.12  ; SE:CP2ﾌﾟﾛｰﾌﾞ下端
AND 13.14  ; SE:CP3ﾌﾟﾛｰﾌﾞ下端
TIMH(015) 0402 #0  ; :
; rung 6
LD T0402  ; :
OUT 402.04  ; 測定動作_C/E
; rung 7
@LD 402.04  ; 測定動作_C/E
OR 403.00  ; 測定終了保持
@ANDNOT 201.05  ; 搬送_搬送位置_GO_OFF
OUT 403.00  ; 測定終了保持

### Section 出力

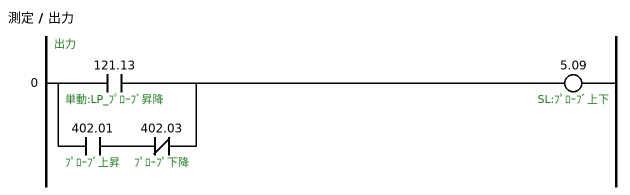
; rung 0: 出力
LD 121.13  ; 単動:LP_ﾌﾟﾛｰﾌﾞ昇降
LD 402.01  ; ﾌﾟﾛｰﾌﾞ上昇
ANDNOT 402.03  ; ﾌﾟﾛｰﾌﾟ下降
ORLD
OUT 5.09  ; SL:ﾌﾟﾛｰﾌﾞ上下

### Section ｴﾗｰ

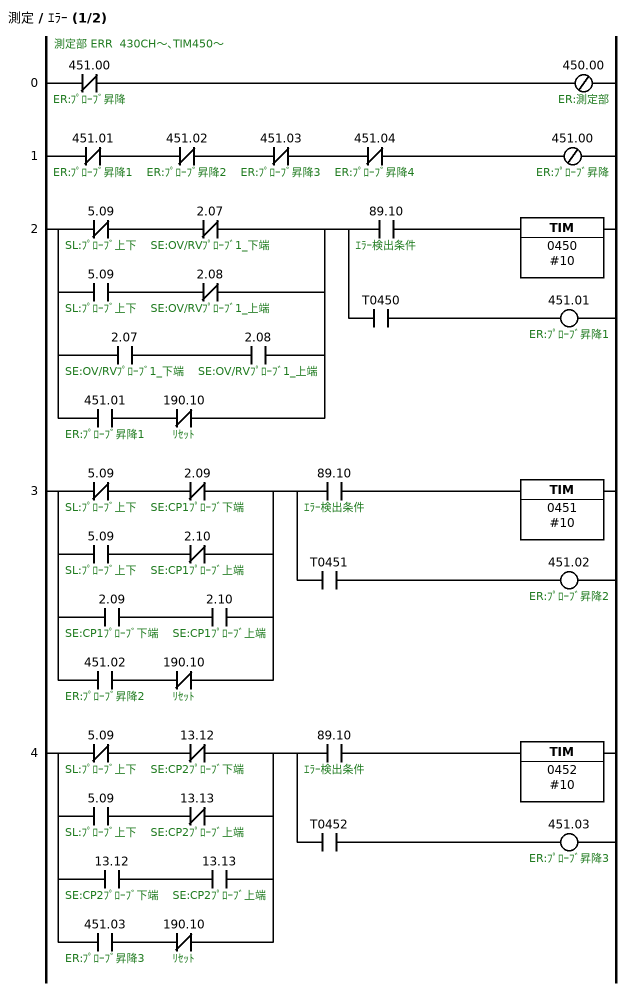
; rung 0: 測定部 ERR  430CH～､TIM450～
LDNOT 451.00  ; ER:ﾌﾟﾛｰﾌﾞ昇降
OUTNOT 450.00  ; ER:測定部
; rung 1
LDNOT 451.01  ; ER:ﾌﾟﾛｰﾌﾞ昇降1
ANDNOT 451.02  ; ER:ﾌﾟﾛｰﾌﾞ昇降2
ANDNOT 451.03  ; ER:ﾌﾟﾛｰﾌﾞ昇降3
ANDNOT 451.04  ; ER:ﾌﾟﾛｰﾌﾞ昇降4
OUTNOT 451.00  ; ER:ﾌﾟﾛｰﾌﾞ昇降
; rung 2
LDNOT 5.09  ; SL:ﾌﾟﾛｰﾌﾞ上下
ANDNOT 2.07  ; SE:OV/RVﾌﾟﾛｰﾌﾞ1_下端
LD 5.09  ; SL:ﾌﾟﾛｰﾌﾞ上下
ANDNOT 2.08  ; SE:OV/RVﾌﾟﾛｰﾌﾞ1_上端
ORLD
LD 2.07  ; SE:OV/RVﾌﾟﾛｰﾌﾞ1_下端
AND 2.08  ; SE:OV/RVﾌﾟﾛｰﾌﾞ1_上端
ORLD
LD 451.01  ; ER:ﾌﾟﾛｰﾌﾞ昇降1
ANDNOT 190.10  ; ﾘｾｯﾄ
ORLD
OUT TR0
AND 89.10  ; ｴﾗｰ検出条件
TIM 0450 #10
LD TR0
AND T0450
OUT 451.01  ; ER:ﾌﾟﾛｰﾌﾞ昇降1
; rung 3
LDNOT 5.09  ; SL:ﾌﾟﾛｰﾌﾞ上下
ANDNOT 2.09  ; SE:CP1ﾌﾟﾛｰﾌﾞ下端
LD 5.09  ; SL:ﾌﾟﾛｰﾌﾞ上下
ANDNOT 2.10  ; SE:CP1ﾌﾟﾛｰﾌﾞ上端
ORLD
LD 2.09  ; SE:CP1ﾌﾟﾛｰﾌﾞ下端
AND 2.10  ; SE:CP1ﾌﾟﾛｰﾌﾞ上端
ORLD
LD 451.02  ; ER:ﾌﾟﾛｰﾌﾞ昇降2
ANDNOT 190.10  ; ﾘｾｯﾄ
ORLD
OUT TR0
AND 89.10  ; ｴﾗｰ検出条件
TIM 0451 #10
LD TR0
AND T0451
OUT 451.02  ; ER:ﾌﾟﾛｰﾌﾞ昇降2
; rung 4
LDNOT 5.09  ; SL:ﾌﾟﾛｰﾌﾞ上下
ANDNOT 13.12  ; SE:CP2ﾌﾟﾛｰﾌﾞ下端
LD 5.09  ; SL:ﾌﾟﾛｰﾌﾞ上下
ANDNOT 13.13  ; SE:CP2ﾌﾟﾛｰﾌﾞ上端
ORLD
LD 13.12  ; SE:CP2ﾌﾟﾛｰﾌﾞ下端
AND 13.13  ; SE:CP2ﾌﾟﾛｰﾌﾞ上端
ORLD
LD 451.03  ; ER:ﾌﾟﾛｰﾌﾞ昇降3
ANDNOT 190.10  ; ﾘｾｯﾄ
ORLD
OUT TR0
AND 89.10  ; ｴﾗｰ検出条件
TIM 0452 #10
LD TR0
AND T0452
OUT 451.03  ; ER:ﾌﾟﾛｰﾌﾞ昇降3

